Universal Robots PolyScope program: 6exPoseList.urp

Program 6exPoseList (installation=default directory=/home/ur/ursim-current/programs createdIn=5.11.8.1010444 lastSavedIn=5.11.8.1010444 robotSerialNumber=20195399999)
Calibrated DH parameters: a=[0, -0.24355, -0.2132, 0, 0, 0]; d=[0.15185, 0, 0, 0.13105, 0.08535, 0.0921]; alpha=[1.570796, 0, 0, 1.570796, -1.570796, 0]; deltaTheta=[0, 0, 0, 0, 0, 0]
BeforeStart
  Script file /home/ur/ursim-current/programs/Script/6_ex_Going_Though_a_list_of_poses.script
    | def MoveLinear(pose_x0, pose_x1):
    | 	i = 0
    | 	while i < 6:
    | 		movel(pose_x0[i], accel_mss, speed_ms, blend_radius_m)
    | 		 sleep (0.5)
    | 		movel(pose_x1[i], accel_mss, speed_ms, blend_radius_m)
    | 		sleep (0.5)
    | 		i = i + 1
    | 	end
    | end
  'Start position'
  x := 0.0
  y := -0.35
  z := 0.3
  rx := 0
  ry := 3.14
  rz := 0
  'going to start position via movej'
  Script: movej(p[x,y,z,rx,ry,rz],a=1,v=1)
Robot Program (runOnlyOnce=false)
  Wait Sleep waitTime=0.01
  accel_mss := 0.3
  speed_ms := 0.3
  blend_radius_m := 0.1
  Call Pose_x0_list_sub
  Call Pose_x1_list_sub
  Script: MoveLinear(pose_x0_list, pose_x1_list)
SubProgram -> Pose_x0_list_sub
SubProgram -> Pose_x1_list_sub
SubProgram Pose_x0_list_sub (keepSynchronizedWithDisk=false)
  pose_1 := p[-0.3,0.3,0.3,3.14,0.0,0.0]
  pose_2 := p[-0.2,0.3,0.3,3.14,0.0,0.0]
  pose_3 := p[-0.1,0.3,0.3,3.14,0.0,0.0]
  pose_4 := p[0.0,0.3,0.3,3.14,0.0,0.0]
  pose_5 := p[0.1,0.3,0.3,3.14,0.0,0.0]
  pose_6 := p[0.2,0.3,0.3,3.14,0.0,0.0]
  pose_x0_list := [pose_1, pose_2, pose_3, pose_4, pose_5, pose_6]
SubProgram Pose_x1_list_sub (keepSynchronizedWithDisk=false)
  pose_01 := p[-0.3,0.2,0.3,3.14,0.0,0.0]
  pose_02 := p[-0.2,0.2,0.3,3.14,0.0,0.0]
  pose_03 := p[-0.1,0.2,0.3,3.14,0.0,0.0]
  pose_04 := p[0.0,0.2,0.3,3.14,0.0,0.0]
  pose_05 := p[0.1,0.2,0.3,3.14,0.0,0.0]
  pose_06 := p[0.2,0.2,0.3,3.14,0.0,0.0]
  pose_x1_list := [pose_01, pose_02, pose_03, pose_04, pose_05, pose_06]
